FUNCTION_BLOCK itfScaleAnalogOutputImplement EXTENDS itfScaleAnalogInputImplement
VAR_INPUT
END_VAR
VAR_OUTPUT
END_VAR
VAR
END_VAR

METHOD mScale : INT
pScaledSignal := pAnalogSignal * pMaxSignalValue;
END_METHOD

END_FUNCTION_BLOCK

(* stored: Version 1.1.0.1, ProductVersion 3.1.4024.12
   POU itfScaleAnalogOutputImplement: Id {0baff21a-3862-4853-9d3f-1bc9f74a7499}, SpecialFunc None
   Method mScale: Id {ba3ea907-ba65-4be2-9d71-8a3ab086a4b8} *)
